Fanuc KAREL source: kb00176.KL

-- PROVISIONAL review KL for V770-1; original PC SHA256 8161b89f5911d42dd498387df239ac2cca81e664c7a9b7ebb178849ffa6397c7
-- Incomplete behavior may be omitted. Consult companion uncertainty JSON. Do not deploy.
PROGRAM KB00176
%NOLOCKGROUP
BEGIN
  -- UNRESOLVED_PC offsets 5-12; opcodes 9D,23
  -- UNRESOLVED_PC offsets 17-32; opcodes 2E,22,32,35
  -- UNRESOLVED_PC offsets 37-44; opcodes 9D,23
  -- UNRESOLVED_PC offsets 49-79; opcodes 27,22,22,1C,22,27,9D,31
  -- UNRESOLVED_PC offsets 84-88; opcodes 7F
END KB00176
